(*
    Handle positive/negative backlash compensation
    User needs to set the direction of backlash from the sign of the compensation value
    Backlash compensation is disabled during referencing (homing).
    When direction is positive/negative, further movement in the negative/positive direction not compensated
    further movement in the negative/positive direction will be compensated
*)
FUNCTION_BLOCK FB_BacklashCompensationNC IMPLEMENTS I_BacklashCompensation
VAR
    {attribute 'no_copy'}
    AxisRef : REFERENCE TO AXIS_REF;
	iMotionLogger : I_MotionLogger := 0;
    fbMcBacklashCompensation: MC_BacklashCompensation;
    (* Other status information for users of the IOC *)
    // Enabled axis backlash compensation
    {attribute 'pytmc' := '
        pv: PLC:bBacklashEnable
        io: io
        field: ZNAM FALSE
        field: ONAM TRUE
        field: DESC Enable Backlash compensation
    '}
    bBacklashEnable: BOOL;

    // backlash compensation status
    {attribute 'pytmc' := '
        pv: PLC:bBacklashStatus
        io: i
        field: ZNAM DISABLED
        field: ONAM ENABLED
        field: DESC Backlash compensation status
    '}
    bBacklashStatus: BOOL;

    // Backlash compensation value
    {attribute 'pytmc' := '
        pv: PLC:fBacklashComp
        io: io
        field: DESC Backlash compensation
    '}
    fBacklash: LREAL := 0.0;

    // Backlash Ramp Velocity
    {attribute 'pytmc' := '
        pv: PLC:fRampVelo
        io: io
        field: DESC Backlash compensation Ramp Velocity
    '}
     fRampVelo : LREAL := 0.0;

    // Current Backlash compensation value ?
    {attribute 'pytmc' := '
        pv: PLC:fMeasuredBacklashComp
        io: i
        field: DESC Currently applied compensation
    '}
    fCurrentBacklash: LREAL;
    {attribute 'hide'}
    fCurrentCompensation : LREAL := 0.0;
    {attribute 'hide'}
    bEnable: BOOL;
    {attribute 'hide'}
    rtbacklashCompensation : R_TRIG;
    {attribute 'hide'}
    bLocalEnable : BOOL;
    {attribute 'hide'}
    sMessage : T_MAXSTRING;
END_VAR

IF NOT __ISVALIDREF(AxisRef) THEN
    RETURN;
END_IF

AxisRef.ReadStatus();
// Monitor EPICS interface and reset to register a new compensation value.

rtbacklashCompensation(CLK:=((fBacklash<>fCurrentCompensation) AND AxisRef.Status.NotMoving));
IF 	rtbacklashCompensation.Q THEN
    bEnable := FALSE;
END_IF

fbMcBacklashCompensation( Axis:=AxisRef,
    Enable:=bEnable AND bBacklashEnable,
    Backlash:= fBacklash,
    CompensationInPositiveDirection:=(fBacklash < 0.0),
    Ramp:=fRampVelo,
    DisableMode	:= E_DISABLEMODE.DisableModeReset,
);
fCurrentCompensation := fBacklash;

IF fbMcBacklashCompensation.Error THEN
	iMotionLogger.Logger(Message := iMotionLogger.ErrorCodeLookup(fbMcBacklashCompensation.ErrorID), Level := E_MotionLogLevel.ERROR, Source := 'BacklashCompensation');	
END_IF

METHOD BacklashCompensation
VAR_INPUT
    Enable	: BOOL := FALSE;
    RampVelo	: LREAL;
END_VAR
THIS^.bEnable := Enable AND THIS^.bBacklashEnable;
THIS^.fRampVelo := RampVelo;

fbMcBacklashCompensation( Axis:=THIS^.AxisRef,
    Enable:=THIS^.bEnable,
    Ramp:=THIS^.fRampVelo,
);
END_METHOD

PROPERTY Busy : BOOL
GET
Busy := fbMcBacklashCompensation.Busy;
END_GET
END_PROPERTY

METHOD PUBLIC CallAfterInit
VAR_INPUT
    AxisRef : REFERENCE TO AXIS_REF;
	iMotionLogger : I_MotionLogger;
END_VAR
THIS^.AxisRef REF= AxisRef;
THIS^.iMotionLogger := iMotionLogger;
END_METHOD

PROPERTY CurrentBacklash : LREAL
GET
END_GET
END_PROPERTY

(*DO NOT use in production code.*)
METHOD EnableBacklashCompensation
VAR_INPUT
    UserEnable : BOOL;
    Compensation : LREAL;
END_VAR
THIS^.bBacklashEnable := UserEnable;
THIS^.fBacklash := Compensation;

fbMcBacklashCompensation( Axis:=AxisRef,
    Enable:= FALSE,
    Backlash:=Compensation
);
END_METHOD

PROPERTY Error : BOOL
GET
Error := THIS^.fbMcBacklashCompensation.Error;
END_GET
END_PROPERTY

PROPERTY ErrorID : UDINT
GET
ErrorID := THIS^.fbMcBacklashCompensation.ErrorID;
END_GET
END_PROPERTY

METHOD FB_Init : BOOL
VAR_INPUT
    bInitRetains : BOOL; // if TRUE, the retain variables are initialized (warm start / cold start)
    bInCopyCode : BOOL;  // if TRUE, the instance afterwards gets moved into the copy code (online change)
    AxisRef : REFERENCE TO AXIS_REF;
	iMotionLogger : I_MotionLogger;
END_VAR
THIS^.AxisRef REF= AxisRef;
THIS^.iMotionLogger := iMotionLogger;
END_METHOD

PROPERTY Message : T_MaxString
GET
Message :=sMessage;
END_GET
END_PROPERTY

PROPERTY Status : BOOL
GET
status := fbMcBacklashCompensation.Enabled;
END_GET
END_PROPERTY

END_FUNCTION_BLOCK

(* stored: Version 1.1.0.1
   POU FB_BacklashCompensationNC: Id {15421978-726d-43ca-8e30-d33510c30e01}, SpecialFunc None
   Method BacklashCompensation: Id {72d6dae3-a62a-450e-865b-c60a18c47466}
   Property Busy: Id {67db6598-5154-4b86-b034-ccf5383284d7}
   Get Get: Id {1e5680ce-0bf7-483a-a265-b25d19a5fa6c}
   Method CallAfterInit: Id {59b21a6b-3d1b-46f2-866a-5384398ac207}
   Property CurrentBacklash: Id {cbe427fc-3f49-4b37-9ce2-197f792afdcd}
   Get Get: Id {c8ce09c0-5517-4ca5-b11a-a6e73bcf0046}
   Method EnableBacklashCompensation: Id {5e2ffdc2-d9b7-43ca-8da1-133fa26b619c}
   Property Error: Id {0213434a-d40a-49c7-a6b4-a3e9e9a7a41a}
   Get Get: Id {c1a3c97c-ae91-4276-85b5-feecf9e8d7c5}
   Property ErrorID: Id {b6765fc0-40e7-4ce5-aa13-569ea50920db}
   Get Get: Id {3dbdc77e-7172-4e8a-b541-0b84a6087295}
   Method FB_Init: Id {86eeb26b-dd4d-42ae-bdf4-cda3d947fa1b}
   Property Message: Id {799861dc-10f6-42dd-a8b5-747f46787023}
   Get Get: Id {b04d60be-1e7a-4ed8-aad3-cee013905d08}
   Property Status: Id {9ab725b4-a349-4d8f-bae9-65d83e60c7e9}
   Get Get: Id {ad2b2cf3-4280-4b71-8ab1-cdec9c65c1b4} *)
